// TIA Portal V20 export
TYPE "ROUT_Datos_Lectura_Scanner"
   STRUCT
      Lectura_SCR : Array[0..19] of Char;
   END_STRUCT;
END_TYPE
